INTERFACE I_HE_SATT_FilterConstantThickness EXTENDS I_HE_SATT_Filter

PROPERTY Thickness : LREAL
GET
END_GET
END_PROPERTY

END_INTERFACE

(* stored: Version 1.1.0.1
   Itf I_HE_SATT_FilterConstantThickness: Id {9d932342-e0ca-4906-9116-279ce19d9c00}
   Property Thickness: Id {5d39f9ee-8615-4426-b7c8-f2e4785a0ab4}
   Get Get: Id {d219a0c1-ed05-4429-bacb-2918c10e1377} *)
